FUNCTION_BLOCK UT_ButtonMapping_DOWN (* Service Interface Function Block Type *)
  (* Standard: ISO 11783-6; Classification: Button – ISO 11783-6 – B.7; Function: All Inputs; Type: UT according to ISO 11783-6 *)
  (* Version 1.0, 2018-12-05, Jose Cabral *)
  (* Version 1.0_DOWN, 2022-08-04, Franz Höpfinger, Unknown *)
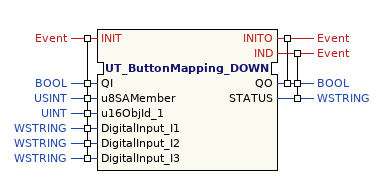
  EVENT_INPUT
    INIT WITH QI, u8SAMember, u16ObjId_1, DigitalInput_I1, DigitalInput_I2, DigitalInput_I3; (* Service Initialization *)
  END_EVENT
  EVENT_OUTPUT
    INITO WITH QO; (* Initialization Confirm *)
    IND WITH QO, STATUS; (* Indication from Resource *)
  END_EVENT
  VAR_INPUT
    QI : BOOL; (* Event Input Qualifier *)
    u8SAMember : USINT := 255; (* Dummy !, set to 255 if in doubt. 0 deactivates FB. *)
    u16ObjId_1 : UINT := 6000; (* Object ID of Input 1 *)
    DigitalInput_I1 : WSTRING := "Button_6000_DOWN"; (* Identifier for Input 1 *)
    DigitalInput_I2 : WSTRING := "Button_6001_DOWN"; (* Identifier for Input 2 *)
    DigitalInput_I3 : WSTRING := "Button_6002_DOWN"; (* Identifier for Input 3 *)
  END_VAR
  VAR_OUTPUT
    QO : BOOL; (* Event Output Qualifier *)
    STATUS : WSTRING; (* Service Status *)
  END_VAR
END_FUNCTION_BLOCK
